FUNCTION_BLOCK Overcurrent_Protector (* Extracted Composite Function Block Type *)
  (* Standard: 61499-2 *)
  (* Version 2/9/2024, Maxth *)
  PACKAGE Main;
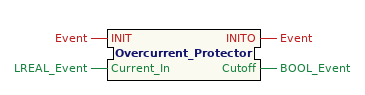
  EVENT_INPUT
    INIT;
  END_EVENT
  EVENT_OUTPUT
    INITO;
  END_EVENT
  SOCKETS
    Current_In : LREAL_Event;
  END_SOCKETS
  PLUGS
    Cutoff : BOOL_Event;
  END_PLUGS
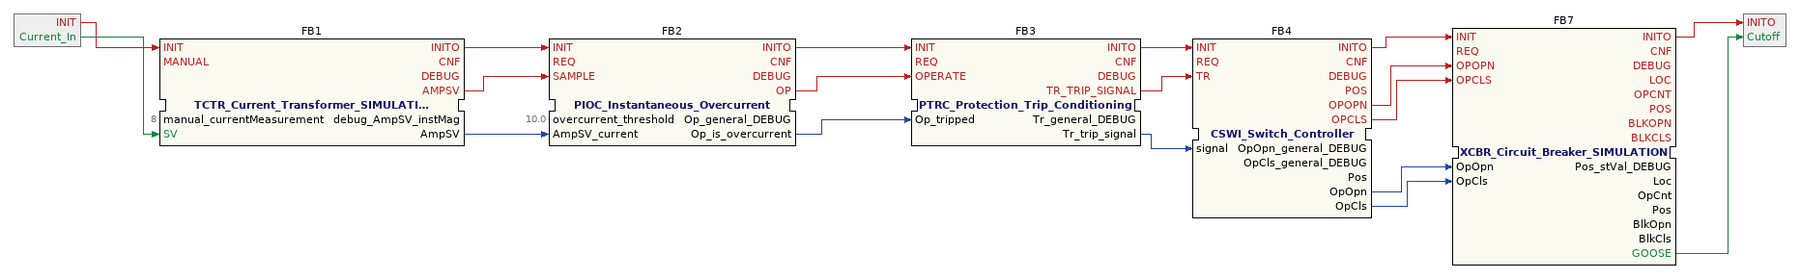
  FBS
    FB1 : TCTR_Current_Transformer_SIMULATION(manual_currentMeasurement := 8);
    FB2 : PIOC_Instantaneous_Overcurrent(overcurrent_threshold := 10.0);
    FB3 : PTRC_Protection_Trip_Conditioning;
    FB4 : CSWI_Switch_Controller;
    FB7 : XCBR_Circuit_Breaker_SIMULATION;
  END_FBS
  EVENT_CONNECTIONS
    FB1.INITO TO FB2.INIT;
    FB1.AMPSV TO FB2.SAMPLE;
    FB2.INITO TO FB3.INIT;
    FB2.OP TO FB3.OPERATE;
    FB3.INITO TO FB4.INIT;
    FB3.TR_TRIP_SIGNAL TO FB4.TR;
    FB4.INITO TO FB7.INIT;
    FB4.OPOPN TO FB7.OPOPN;
    FB4.OPCLS TO FB7.OPCLS;
    INIT TO FB1.INIT;
    FB7.INITO TO INITO;
  END_CONNECTIONS
  DATA_CONNECTIONS
    FB1.AmpSV TO FB2.AmpSV_current;
    FB2.Op_is_overcurrent TO FB3.Op_tripped;
    FB3.Tr_trip_signal TO FB4.signal;
    FB4.OpOpn TO FB7.OpOpn;
    FB4.OpCls TO FB7.OpCls;
  END_CONNECTIONS
  ADAPTER_CONNECTIONS
    Current_In TO FB1.SV;
    FB7.GOOSE TO Cutoff;
  END_CONNECTIONS
END_FUNCTION_BLOCK
